# B&R Automation Studio project BatteryControl (part 4)

```iecst
	sustainHF[0]:=50.000;
	sustainHF[1]:=50.000;
	sustainHF[2]:=50.000;
	sustainHF[3]:=50.000;
	sustainHF[4]:=50.000;
	sustainHF[5]:=50.000;
	sustainHF[6]:=50.000;
	sustainHF[7]:=50.000;
	sustainHF[8]:=50.000;
	sustainHF[9]:=50.000;
	sustainHF[10]:=50.000;
	sustainHF[11]:=50.000;
	sustainHF[12]:=50.000;
	sustainHF[13]:=50.000;
	sustainHF[14]:=50.000;
	sustainHF[15]:=50.000;
	sustainHF[16]:=50.000;
	sustainHF[17]:=50.000;
	sustainHF[18]:=50.000;
	sustainHF[19]:=50.000;
	sustainHF[20]:=50.000;
	sustainHF[21]:=50.000;
	sustainHF[22]:=50.000;
	sustainHF[23]:=50.000;
	sustainHF[24]:=50.000;
	sustainHF[25]:=50.000;
	sustainHF[26]:=50.000;
	sustainHF[27]:=50.000;
	sustainHF[28]:=50.000;
	sustainHF[29]:=50.000;
	sustainHF[30]:=50.600;
	sustainHF[31]:=50.600;
	sustainHF[32]:=50.600;
	sustainHF[33]:=50.600;
	sustainHF[34]:=50.600;
	sustainHF[35]:=50.600;
	sustainHF[36]:=50.600;
	sustainHF[37]:=50.600;
	sustainHF[38]:=50.600;
	sustainHF[39]:=50.600;
	sustainHF[40]:=50.600;
	sustainHF[41]:=50.600;
	sustainHF[42]:=50.600;
	sustainHF[43]:=50.600;
	sustainHF[44]:=50.600;
	sustainHF[45]:=50.600;
	sustainHF[46]:=50.600;
	sustainHF[47]:=50.600;
	sustainHF[48]:=50.600;
	sustainHF[49]:=50.600;
	sustainHF[50]:=50.600;
	sustainHF[51]:=50.600;
	sustainHF[52]:=50.600;
	sustainHF[53]:=50.600;
	sustainHF[54]:=50.600;
	sustainHF[55]:=50.600;
	sustainHF[56]:=50.600;
	sustainHF[57]:=50.600;
	sustainHF[58]:=50.600;
	sustainHF[59]:=50.600;
	sustainHF[60]:=50.600;
	sustainHF[61]:=50.600;
	sustainHF[62]:=50.600;
	sustainHF[63]:=50.600;
	sustainHF[64]:=50.600;
	sustainHF[65]:=50.600;
	sustainHF[66]:=50.600;
	sustainHF[67]:=50.600;
	sustainHF[68]:=50.600;
	sustainHF[69]:=50.600;
	sustainHF[70]:=50.600;
	sustainHF[71]:=50.600;
	sustainHF[72]:=50.600;
	sustainHF[73]:=50.600;
	sustainHF[74]:=50.600;
	sustainHF[75]:=50.600;
	sustainHF[76]:=50.600;
	sustainHF[77]:=50.600;
	sustainHF[78]:=50.600;
	sustainHF[79]:=50.600;
	sustainHF[80]:=50.600;
	sustainHF[81]:=50.600;
	sustainHF[82]:=50.600;
	sustainHF[83]:=50.600;
	sustainHF[84]:=50.600;
	sustainHF[85]:=50.600;
	sustainHF[86]:=50.600;
	sustainHF[87]:=50.600;
	sustainHF[88]:=50.600;
	sustainHF[89]:=50.600;
	sustainHF[90]:=50.600;
	sustainHF[91]:=50.600;
	sustainHF[92]:=50.600;
	sustainHF[93]:=50.600;
	sustainHF[94]:=50.600;
	sustainHF[95]:=50.600;
	sustainHF[96]:=50.600;
	sustainHF[97]:=50.600;
	sustainHF[98]:=50.600;
	sustainHF[99]:=50.600;
	sustainHF[100]:=50.600;
	sustainHF[101]:=50.600;
	sustainHF[102]:=50.600;
	sustainHF[103]:=50.600;
	sustainHF[104]:=50.600;
	sustainHF[105]:=50.600;
	sustainHF[106]:=50.600;
	sustainHF[107]:=50.600;
	sustainHF[108]:=50.600;
	sustainHF[109]:=50.600;
	sustainHF[110]:=50.600;
	sustainHF[111]:=50.600;
	sustainHF[112]:=50.600;
	sustainHF[113]:=50.600;
	sustainHF[114]:=50.600;
	sustainHF[115]:=50.600;
	sustainHF[116]:=50.600;
	sustainHF[117]:=50.600;
	sustainHF[118]:=50.600;
	sustainHF[119]:=50.600;
	sustainHF[120]:=50.600;
	sustainHF[121]:=50.600;
	sustainHF[122]:=50.600;
	sustainHF[123]:=50.600;
	sustainHF[124]:=50.600;
	sustainHF[125]:=50.600;
	sustainHF[126]:=50.600;
	sustainHF[127]:=50.600;
	sustainHF[128]:=50.600;
	sustainHF[129]:=50.600;
	sustainHF[130]:=50.600;
	sustainHF[131]:=50.600;
	sustainHF[132]:=50.600;
	sustainHF[133]:=50.600;
	sustainHF[134]:=50.600;
	sustainHF[135]:=50.600;
	sustainHF[136]:=50.600;
	sustainHF[137]:=50.600;
	sustainHF[138]:=50.600;
	sustainHF[139]:=50.600;
	sustainHF[140]:=50.600;
	sustainHF[141]:=50.600;
	sustainHF[142]:=50.600;
	sustainHF[143]:=50.600;
	sustainHF[144]:=50.600;
	sustainHF[145]:=50.600;
	sustainHF[146]:=50.600;
	sustainHF[147]:=50.600;
	sustainHF[148]:=50.600;
	sustainHF[149]:=50.600;
	sustainHF[150]:=50.600;
	sustainHF[151]:=50.600;
	sustainHF[152]:=50.600;
	sustainHF[153]:=50.600;
	sustainHF[154]:=50.600;
	sustainHF[155]:=50.600;
	sustainHF[156]:=50.600;
	sustainHF[157]:=50.600;
	sustainHF[158]:=50.600;
	sustainHF[159]:=50.600;
	sustainHF[160]:=50.600;
	sustainHF[161]:=50.600;
	sustainHF[162]:=50.600;
	sustainHF[163]:=50.600;
	sustainHF[164]:=50.600;
	sustainHF[165]:=50.600;
	sustainHF[166]:=50.600;
	sustainHF[167]:=50.600;
	sustainHF[168]:=50.600;
	sustainHF[169]:=50.600;
	sustainHF[170]:=50.600;
	sustainHF[171]:=50.600;
	sustainHF[172]:=50.600;
	sustainHF[173]:=50.600;
	sustainHF[174]:=50.600;
	sustainHF[175]:=50.600;
	sustainHF[176]:=50.600;
	sustainHF[177]:=50.600;
	sustainHF[178]:=50.600;
	sustainHF[179]:=50.600;
	sustainHF[180]:=50.600;
	sustainHF[181]:=50.600;
	sustainHF[182]:=50.600;
	sustainHF[183]:=50.600;
	sustainHF[184]:=50.600;
	sustainHF[185]:=50.600;
	sustainHF[186]:=50.600;
	sustainHF[187]:=50.600;
	sustainHF[188]:=50.600;
	sustainHF[189]:=50.600;
	sustainHF[190]:=50.600;
	sustainHF[191]:=50.600;
	sustainHF[192]:=50.600;
	sustainHF[193]:=50.600;
	sustainHF[194]:=50.600;
	sustainHF[195]:=50.600;
	sustainHF[196]:=50.600;
	sustainHF[197]:=50.600;
	sustainHF[198]:=50.600;
	sustainHF[199]:=50.600;
	sustainHF[200]:=50.600;
	sustainHF[201]:=50.600;
	sustainHF[202]:=50.600;
	sustainHF[203]:=50.600;
	sustainHF[204]:=50.600;
	sustainHF[205]:=50.600;
	sustainHF[206]:=50.600;
	sustainHF[207]:=50.600;
	sustainHF[208]:=50.600;
	sustainHF[209]:=50.600;
	sustainHF[210]:=50.600;
	sustainHF[211]:=50.600;
	sustainHF[212]:=50.600;
	sustainHF[213]:=50.600;
	sustainHF[214]:=50.600;
	sustainHF[215]:=50.600;
	sustainHF[216]:=50.600;
	sustainHF[217]:=50.600;
	sustainHF[218]:=50.600;
	sustainHF[219]:=50.600;
	sustainHF[220]:=50.600;
	sustainHF[221]:=50.600;
	sustainHF[222]:=50.600;
	sustainHF[223]:=50.600;
	sustainHF[224]:=50.600;
	sustainHF[225]:=50.600;
	sustainHF[226]:=50.600;
	sustainHF[227]:=50.600;
	sustainHF[228]:=50.600;
	sustainHF[229]:=50.600;
	sustainHF[230]:=50.600;
	sustainHF[231]:=50.600;
	sustainHF[232]:=50.600;
	sustainHF[233]:=50.600;
	sustainHF[234]:=50.600;
	sustainHF[235]:=50.600;
	sustainHF[236]:=50.600;
	sustainHF[237]:=50.600;
	sustainHF[238]:=50.600;
	sustainHF[239]:=50.600;
	sustainHF[240]:=50.600;
	sustainHF[241]:=50.600;
	sustainHF[242]:=50.600;
	sustainHF[243]:=50.600;
	sustainHF[244]:=50.600;
	sustainHF[245]:=50.600;
	sustainHF[246]:=50.600;
	sustainHF[247]:=50.600;
	sustainHF[248]:=50.600;
	sustainHF[249]:=50.600;
	sustainHF[250]:=50.600;
	sustainHF[251]:=50.600;
	sustainHF[252]:=50.600;
	sustainHF[253]:=50.600;
	sustainHF[254]:=50.600;
	sustainHF[255]:=50.600;
	sustainHF[256]:=50.600;
	sustainHF[257]:=50.600;
	sustainHF[258]:=50.600;
	sustainHF[259]:=50.600;
	sustainHF[260]:=50.600;
	sustainHF[261]:=50.600;
	sustainHF[262]:=50.600;
	sustainHF[263]:=50.600;
	sustainHF[264]:=50.600;
	sustainHF[265]:=50.600;
	sustainHF[266]:=50.600;
	sustainHF[267]:=50.600;
	sustainHF[268]:=50.600;
	sustainHF[269]:=50.600;
	sustainHF[270]:=50.600;
	sustainHF[271]:=50.600;
	sustainHF[272]:=50.600;
	sustainHF[273]:=50.600;
	sustainHF[274]:=50.600;
	sustainHF[275]:=50.600;
	sustainHF[276]:=50.600;
	sustainHF[277]:=50.600;
	sustainHF[278]:=50.600;
	sustainHF[279]:=50.600;
	sustainHF[280]:=50.600;
	sustainHF[281]:=50.600;
	sustainHF[282]:=50.600;
	sustainHF[283]:=50.600;
	sustainHF[284]:=50.600;
	sustainHF[285]:=50.600;
	sustainHF[286]:=50.600;
	sustainHF[287]:=50.600;
	sustainHF[288]:=50.600;
	sustainHF[289]:=50.600;
	sustainHF[290]:=50.600;
	sustainHF[291]:=50.600;
	sustainHF[292]:=50.600;
	sustainHF[293]:=50.600;
	sustainHF[294]:=50.600;
	sustainHF[295]:=50.600;
	sustainHF[296]:=50.600;
	sustainHF[297]:=50.600;
	sustainHF[298]:=50.600;
	sustainHF[299]:=50.600;
	sustainHF[300]:=50.600;
	sustainHF[301]:=50.600;
	sustainHF[302]:=50.600;
	sustainHF[303]:=50.600;
	sustainHF[304]:=50.600;
	sustainHF[305]:=50.600;
	sustainHF[306]:=50.600;
	sustainHF[307]:=50.600;
	sustainHF[308]:=50.600;
	sustainHF[309]:=50.600;
	sustainHF[310]:=50.600;
	sustainHF[311]:=50.600;
	sustainHF[312]:=50.600;
	sustainHF[313]:=50.600;
	sustainHF[314]:=50.600;
	sustainHF[315]:=50.600;
	sustainHF[316]:=50.600;
	sustainHF[317]:=50.600;
	sustainHF[318]:=50.600;
	sustainHF[319]:=50.600;
	sustainHF[320]:=50.600;
	sustainHF[321]:=50.600;
	sustainHF[322]:=50.600;
	sustainHF[323]:=50.600;
	sustainHF[324]:=50.600;
	sustainHF[325]:=50.600;
	sustainHF[326]:=50.600;
	sustainHF[327]:=50.600;
	sustainHF[328]:=50.600;
	sustainHF[329]:=50.600;
	sustainHF[330]:=50.600;
	sustainHF[331]:=50.600;
	sustainHF[332]:=50.600;
	sustainHF[333]:=50.600;
	sustainHF[334]:=50.600;
	sustainHF[335]:=50.600;
	sustainHF[336]:=50.600;
	sustainHF[337]:=50.600;
	sustainHF[338]:=50.600;
	sustainHF[339]:=50.600;
	sustainHF[340]:=50.600;
	sustainHF[341]:=50.600;
	sustainHF[342]:=50.600;
	sustainHF[343]:=50.600;
	sustainHF[344]:=50.600;
	sustainHF[345]:=50.600;
	sustainHF[346]:=50.600;
	sustainHF[347]:=50.600;
	sustainHF[348]:=50.600;
	sustainHF[349]:=50.600;
	sustainHF[350]:=50.600;
	sustainHF[351]:=50.600;
	sustainHF[352]:=50.600;
	sustainHF[353]:=50.600;
	sustainHF[354]:=50.600;
	sustainHF[355]:=50.600;
	sustainHF[356]:=50.600;
	sustainHF[357]:=50.600;
	sustainHF[358]:=50.600;
	sustainHF[359]:=50.600;
	sustainHF[360]:=50.600;
	sustainHF[361]:=50.600;
	sustainHF[362]:=50.600;
	sustainHF[363]:=50.600;
	sustainHF[364]:=50.600;
	sustainHF[365]:=50.600;
	sustainHF[366]:=50.600;
	sustainHF[367]:=50.600;
	sustainHF[368]:=50.600;
	sustainHF[369]:=50.600;
	sustainHF[370]:=50.600;
	sustainHF[371]:=50.600;
	sustainHF[372]:=50.600;
	sustainHF[373]:=50.600;
	sustainHF[374]:=50.600;
	sustainHF[375]:=50.600;
	sustainHF[376]:=50.600;
	sustainHF[377]:=50.600;
	sustainHF[378]:=50.600;
	sustainHF[379]:=50.600;
	sustainHF[380]:=50.600;
	sustainHF[381]:=50.600;
	sustainHF[382]:=50.600;
	sustainHF[383]:=50.600;
	sustainHF[384]:=50.600;
	sustainHF[385]:=50.600;
	sustainHF[386]:=50.600;
	sustainHF[387]:=50.600;
	sustainHF[388]:=50.600;
	sustainHF[389]:=50.600;
	sustainHF[390]:=50.600;
	sustainHF[391]:=50.600;
	sustainHF[392]:=50.600;
	sustainHF[393]:=50.600;
	sustainHF[394]:=50.600;
	sustainHF[395]:=50.600;
	sustainHF[396]:=50.600;
	sustainHF[397]:=50.600;
	sustainHF[398]:=50.600;
	sustainHF[399]:=50.600;
	sustainHF[400]:=50.600;
	sustainHF[401]:=50.600;
	sustainHF[402]:=50.600;
	sustainHF[403]:=50.600;
	sustainHF[404]:=50.600;
	sustainHF[405]:=50.600;
	sustainHF[406]:=50.600;
	sustainHF[407]:=50.600;
	sustainHF[408]:=50.600;
	sustainHF[409]:=50.600;
	sustainHF[410]:=50.600;
	sustainHF[411]:=50.600;
	sustainHF[412]:=50.600;
	sustainHF[413]:=50.600;
	sustainHF[414]:=50.600;
	sustainHF[415]:=50.600;
	sustainHF[416]:=50.600;
	sustainHF[417]:=50.600;
	sustainHF[418]:=50.600;
	sustainHF[419]:=50.600;
	sustainHF[420]:=50.600;
	sustainHF[421]:=50.600;
	sustainHF[422]:=50.600;
	sustainHF[423]:=50.600;
	sustainHF[424]:=50.600;
	sustainHF[425]:=50.600;
	sustainHF[426]:=50.600;
	sustainHF[427]:=50.600;
	sustainHF[428]:=50.600;
	sustainHF[429]:=50.600;
	sustainHF[430]:=50.600;
	sustainHF[431]:=50.600;
	sustainHF[432]:=50.600;
	sustainHF[433]:=50.600;
	sustainHF[434]:=50.600;
	sustainHF[435]:=50.600;
	sustainHF[436]:=50.600;
	sustainHF[437]:=50.600;
	sustainHF[438]:=50.600;
	sustainHF[439]:=50.600;
	sustainHF[440]:=50.600;
	sustainHF[441]:=50.600;
	sustainHF[442]:=50.600;
	sustainHF[443]:=50.600;
	sustainHF[444]:=50.600;
	sustainHF[445]:=50.600;
	sustainHF[446]:=50.600;
	sustainHF[447]:=50.600;
	sustainHF[448]:=50.600;
	sustainHF[449]:=50.600;
	sustainHF[450]:=50.600;
	sustainHF[451]:=50.600;
	sustainHF[452]:=50.600;
	sustainHF[453]:=50.600;
	sustainHF[454]:=50.600;
	sustainHF[455]:=50.600;
	sustainHF[456]:=50.600;
	sustainHF[457]:=50.600;
	sustainHF[458]:=50.600;
	sustainHF[459]:=50.600;
	sustainHF[460]:=50.600;
	sustainHF[461]:=50.600;
	sustainHF[462]:=50.600;
	sustainHF[463]:=50.600;
	sustainHF[464]:=50.600;
	sustainHF[465]:=50.600;
	sustainHF[466]:=50.600;
	sustainHF[467]:=50.600;
	sustainHF[468]:=50.600;
	sustainHF[469]:=50.600;
	sustainHF[470]:=50.600;
	sustainHF[471]:=50.600;
	sustainHF[472]:=50.600;
	sustainHF[473]:=50.600;
	sustainHF[474]:=50.600;
	sustainHF[475]:=50.600;
	sustainHF[476]:=50.600;
	sustainHF[477]:=50.600;
	sustainHF[478]:=50.600;
	sustainHF[479]:=50.600;
	sustainHF[480]:=50.600;
	sustainHF[481]:=50.600;
	sustainHF[482]:=50.600;
	sustainHF[483]:=50.600;
	sustainHF[484]:=50.600;
	sustainHF[485]:=50.600;
	sustainHF[486]:=50.600;
	sustainHF[487]:=50.600;
	sustainHF[488]:=50.600;
	sustainHF[489]:=50.600;
	sustainHF[490]:=50.600;
	sustainHF[491]:=50.600;
	sustainHF[492]:=50.600;
	sustainHF[493]:=50.600;
	sustainHF[494]:=50.600;
	sustainHF[495]:=50.600;
	sustainHF[496]:=50.600;
	sustainHF[497]:=50.600;
	sustainHF[498]:=50.600;
	sustainHF[499]:=50.600;
	sustainHF[500]:=50.600;
	sustainHF[501]:=50.600;
	sustainHF[502]:=50.600;
	sustainHF[503]:=50.600;
	sustainHF[504]:=50.600;
	sustainHF[505]:=50.600;
	sustainHF[506]:=50.600;
	sustainHF[507]:=50.600;
	sustainHF[508]:=50.600;
	sustainHF[509]:=50.600;
	sustainHF[510]:=50.600;
	sustainHF[511]:=50.600;
	sustainHF[512]:=50.600;
	sustainHF[513]:=50.600;
	sustainHF[514]:=50.600;
	sustainHF[515]:=50.600;
	sustainHF[516]:=50.600;
	sustainHF[517]:=50.600;
	sustainHF[518]:=50.600;
	sustainHF[519]:=50.600;
	sustainHF[520]:=50.600;
	sustainHF[521]:=50.600;
	sustainHF[522]:=50.600;
	sustainHF[523]:=50.600;
	sustainHF[524]:=50.600;
	sustainHF[525]:=50.600;
	sustainHF[526]:=50.600;
	sustainHF[527]:=50.600;
	sustainHF[528]:=50.600;
	sustainHF[529]:=50.600;
	sustainHF[530]:=50.600;
	sustainHF[531]:=50.600;
	sustainHF[532]:=50.600;
	sustainHF[533]:=50.600;
	sustainHF[534]:=50.600;
	sustainHF[535]:=50.600;
	sustainHF[536]:=50.600;
	sustainHF[537]:=50.600;
	sustainHF[538]:=50.600;
	sustainHF[539]:=50.600;
	sustainHF[540]:=50.600;
	sustainHF[541]:=50.600;
	sustainHF[542]:=50.600;
	sustainHF[543]:=50.600;
	sustainHF[544]:=50.600;
	sustainHF[545]:=50.600;
	sustainHF[546]:=50.600;
	sustainHF[547]:=50.600;
	sustainHF[548]:=50.600;
	sustainHF[549]:=50.600;
	sustainHF[550]:=50.600;
	sustainHF[551]:=50.600;
	sustainHF[552]:=50.600;
	sustainHF[553]:=50.600;
	sustainHF[554]:=50.600;
	sustainHF[555]:=50.600;
	sustainHF[556]:=50.600;
	sustainHF[557]:=50.600;
	sustainHF[558]:=50.600;
	sustainHF[559]:=50.600;
	sustainHF[560]:=50.600;
	sustainHF[561]:=50.600;
	sustainHF[562]:=50.600;
	sustainHF[563]:=50.600;
	sustainHF[564]:=50.600;
	sustainHF[565]:=50.600;
	sustainHF[566]:=50.600;
	sustainHF[567]:=50.600;
	sustainHF[568]:=50.600;
	sustainHF[569]:=50.600;
	sustainHF[570]:=50.600;
	sustainHF[571]:=50.600;
	sustainHF[572]:=50.600;
	sustainHF[573]:=50.600;
	sustainHF[574]:=50.600;
	sustainHF[575]:=50.600;
	sustainHF[576]:=50.600;
	sustainHF[577]:=50.600;
	sustainHF[578]:=50.600;
	sustainHF[579]:=50.600;
	sustainHF[580]:=50.600;
	sustainHF[581]:=50.600;
	sustainHF[582]:=50.600;
	sustainHF[583]:=50.600;
	sustainHF[584]:=50.600;
	sustainHF[585]:=50.600;
	sustainHF[586]:=50.600;
	sustainHF[587]:=50.600;
	sustainHF[588]:=50.600;
	sustainHF[589]:=50.600;
	sustainHF[590]:=50.600;
	sustainHF[591]:=50.600;
	sustainHF[592]:=50.600;
	sustainHF[593]:=50.600;
	sustainHF[594]:=50.600;
	sustainHF[595]:=50.600;
	sustainHF[596]:=50.600;
	sustainHF[597]:=50.600;
	sustainHF[598]:=50.600;
	sustainHF[599]:=50.600;
	sustainHF[600]:=50.600;
	sustainHF[601]:=50.600;
	sustainHF[602]:=50.600;
	sustainHF[603]:=50.600;
	sustainHF[604]:=50.600;
	sustainHF[605]:=50.600;
	sustainHF[606]:=50.600;
	sustainHF[607]:=50.600;
	sustainHF[608]:=50.600;
	sustainHF[609]:=50.600;
	sustainHF[610]:=50.600;
	sustainHF[611]:=50.600;
	sustainHF[612]:=50.600;
	sustainHF[613]:=50.600;
	sustainHF[614]:=50.600;
	sustainHF[615]:=50.600;
	sustainHF[616]:=50.600;
	sustainHF[617]:=50.600;
	sustainHF[618]:=50.600;
	sustainHF[619]:=50.600;
	sustainHF[620]:=50.600;
	sustainHF[621]:=50.600;
	sustainHF[622]:=50.600;
	sustainHF[623]:=50.600;
	sustainHF[624]:=50.600;
	sustainHF[625]:=50.600;
	sustainHF[626]:=50.600;
	sustainHF[627]:=50.600;
	sustainHF[628]:=50.600;
	sustainHF[629]:=50.600;
	sustainHF[630]:=50.600;
	sustainHF[631]:=50.600;
	sustainHF[632]:=50.600;
	sustainHF[633]:=50.600;
	sustainHF[634]:=50.600;
	sustainHF[635]:=50.600;
	sustainHF[636]:=50.600;
	sustainHF[637]:=50.600;
	sustainHF[638]:=50.600;
	sustainHF[639]:=50.600;
	sustainHF[640]:=50.600;
	sustainHF[641]:=50.600;
	sustainHF[642]:=50.600;
	sustainHF[643]:=50.600;
	sustainHF[644]:=50.600;
	sustainHF[645]:=50.600;
	sustainHF[646]:=50.600;
	sustainHF[647]:=50.600;
	sustainHF[648]:=50.600;
	sustainHF[649]:=50.600;
	sustainHF[650]:=50.600;
	sustainHF[651]:=50.600;
	sustainHF[652]:=50.600;
	sustainHF[653]:=50.600;
	sustainHF[654]:=50.600;
	sustainHF[655]:=50.600;
	sustainHF[656]:=50.600;
	sustainHF[657]:=50.600;
	sustainHF[658]:=50.600;
	sustainHF[659]:=50.600;
	sustainHF[660]:=50.600;
	sustainHF[661]:=50.600;
	sustainHF[662]:=50.600;
	sustainHF[663]:=50.600;
	sustainHF[664]:=50.600;
	sustainHF[665]:=50.600;
	sustainHF[666]:=50.600;
	sustainHF[667]:=50.600;
	sustainHF[668]:=50.600;
	sustainHF[669]:=50.600;
	sustainHF[670]:=50.600;
	sustainHF[671]:=50.600;
	sustainHF[672]:=50.600;
	sustainHF[673]:=50.600;
	sustainHF[674]:=50.600;
	sustainHF[675]:=50.600;
	sustainHF[676]:=50.600;
	sustainHF[677]:=50.600;
	sustainHF[678]:=50.600;
	sustainHF[679]:=50.600;
	sustainHF[680]:=50.600;
	sustainHF[681]:=50.600;
	sustainHF[682]:=50.600;
	sustainHF[683]:=50.600;
	sustainHF[684]:=50.600;
	sustainHF[685]:=50.600;
	sustainHF[686]:=50.600;
	sustainHF[687]:=50.600;
	sustainHF[688]:=50.600;
	sustainHF[689]:=50.600;
	sustainHF[690]:=50.600;
	sustainHF[691]:=50.600;
	sustainHF[692]:=50.600;
	sustainHF[693]:=50.600;
	sustainHF[694]:=50.600;
	sustainHF[695]:=50.600;
	sustainHF[696]:=50.600;
	sustainHF[697]:=50.600;
	sustainHF[698]:=50.600;
	sustainHF[699]:=50.600;
	sustainHF[700]:=50.600;
	sustainHF[701]:=50.600;
	sustainHF[702]:=50.600;
	sustainHF[703]:=50.600;
	sustainHF[704]:=50.600;
	sustainHF[705]:=50.600;
	sustainHF[706]:=50.600;
	sustainHF[707]:=50.600;
	sustainHF[708]:=50.600;
	sustainHF[709]:=50.600;
	sustainHF[710]:=50.600;
	sustainHF[711]:=50.600;
	sustainHF[712]:=50.600;
	sustainHF[713]:=50.600;
	sustainHF[714]:=50.600;
	sustainHF[715]:=50.600;
	sustainHF[716]:=50.600;
	sustainHF[717]:=50.600;
	sustainHF[718]:=50.600;
	sustainHF[719]:=50.600;
	sustainHF[720]:=50.600;
	sustainHF[721]:=50.600;
	sustainHF[722]:=50.600;
	sustainHF[723]:=50.600;
	sustainHF[724]:=50.600;
	sustainHF[725]:=50.600;
	sustainHF[726]:=50.600;
	sustainHF[727]:=50.600;
	sustainHF[728]:=50.600;
	sustainHF[729]:=50.600;
	sustainHF[730]:=50.600;
	sustainHF[731]:=50.600;
	sustainHF[732]:=50.600;
	sustainHF[733]:=50.600;
	sustainHF[734]:=50.600;
	sustainHF[735]:=50.600;
	sustainHF[736]:=50.600;
	sustainHF[737]:=50.600;
	sustainHF[738]:=50.600;
	sustainHF[739]:=50.600;
	sustainHF[740]:=50.600;
	sustainHF[741]:=50.600;
	sustainHF[742]:=50.600;
	sustainHF[743]:=50.600;
	sustainHF[744]:=50.600;
	sustainHF[745]:=50.600;
	sustainHF[746]:=50.600;
	sustainHF[747]:=50.600;
	sustainHF[748]:=50.600;
	sustainHF[749]:=50.600;
	sustainHF[750]:=50.600;
	sustainHF[751]:=50.600;
	sustainHF[752]:=50.600;
	sustainHF[753]:=50.600;
	sustainHF[754]:=50.600;
	sustainHF[755]:=50.600;
	sustainHF[756]:=50.600;
	sustainHF[757]:=50.600;
	sustainHF[758]:=50.600;
	sustainHF[759]:=50.600;
	sustainHF[760]:=50.600;
	sustainHF[761]:=50.600;
	sustainHF[762]:=50.600;
	sustainHF[763]:=50.600;
	sustainHF[764]:=50.600;
	sustainHF[765]:=50.600;
	sustainHF[766]:=50.600;
	sustainHF[767]:=50.600;
	sustainHF[768]:=50.600;
	sustainHF[769]:=50.600;
	sustainHF[770]:=50.600;
	sustainHF[771]:=50.600;
	sustainHF[772]:=50.600;
	sustainHF[773]:=50.600;
	sustainHF[774]:=50.600;
	sustainHF[775]:=50.600;
	sustainHF[776]:=50.600;
	sustainHF[777]:=50.600;
	sustainHF[778]:=50.600;
	sustainHF[779]:=50.600;
	sustainHF[780]:=50.600;
	sustainHF[781]:=50.600;
	sustainHF[782]:=50.600;
	sustainHF[783]:=50.600;
	sustainHF[784]:=50.600;
	sustainHF[785]:=50.600;
	sustainHF[786]:=50.600;
	sustainHF[787]:=50.600;
	sustainHF[788]:=50.600;
	sustainHF[789]:=50.600;
	sustainHF[790]:=50.600;
	sustainHF[791]:=50.600;
	sustainHF[792]:=50.600;
	sustainHF[793]:=50.600;
	sustainHF[794]:=50.600;
	sustainHF[795]:=50.600;
	sustainHF[796]:=50.600;
	sustainHF[797]:=50.600;
	sustainHF[798]:=50.600;
	sustainHF[799]:=50.600;
	sustainHF[800]:=50.600;
	sustainHF[801]:=50.600;
	sustainHF[802]:=50.600;
	sustainHF[803]:=50.600;
	sustainHF[804]:=50.600;
	sustainHF[805]:=50.600;
	sustainHF[806]:=50.600;
	sustainHF[807]:=50.600;
	sustainHF[808]:=50.600;
	sustainHF[809]:=50.600;
	sustainHF[810]:=50.600;
	sustainHF[811]:=50.600;
	sustainHF[812]:=50.600;
	sustainHF[813]:=50.600;
	sustainHF[814]:=50.600;
	sustainHF[815]:=50.600;
	sustainHF[816]:=50.600;
	sustainHF[817]:=50.600;
	sustainHF[818]:=50.600;
	sustainHF[819]:=50.600;
	sustainHF[820]:=50.600;
	sustainHF[821]:=50.600;
	sustainHF[822]:=50.600;
	sustainHF[823]:=50.600;
	sustainHF[824]:=50.600;
	sustainHF[825]:=50.600;
	sustainHF[826]:=50.600;
	sustainHF[827]:=50.600;
	sustainHF[828]:=50.600;
	sustainHF[829]:=50.600;
	sustainHF[830]:=50.600;
	sustainHF[831]:=50.600;
	sustainHF[832]:=50.600;
	sustainHF[833]:=50.600;
	sustainHF[834]:=50.600;
	sustainHF[835]:=50.600;
	sustainHF[836]:=50.600;
	sustainHF[837]:=50.600;
	sustainHF[838]:=50.600;
	sustainHF[839]:=50.600;
	sustainHF[840]:=50.600;
	sustainHF[841]:=50.600;
	sustainHF[842]:=50.600;
	sustainHF[843]:=50.600;
	sustainHF[844]:=50.600;
	sustainHF[845]:=50.600;
	sustainHF[846]:=50.600;
	sustainHF[847]:=50.600;
	sustainHF[848]:=50.600;
	sustainHF[849]:=50.600;
	sustainHF[850]:=50.600;
	sustainHF[851]:=50.600;
	sustainHF[852]:=50.600;
	sustainHF[853]:=50.600;
	sustainHF[854]:=50.600;
	sustainHF[855]:=50.600;
	sustainHF[856]:=50.600;
	sustainHF[857]:=50.600;
	sustainHF[858]:=50.600;
	sustainHF[859]:=50.600;
	sustainHF[860]:=50.600;
	sustainHF[861]:=50.600;
	sustainHF[862]:=50.600;
	sustainHF[863]:=50.600;
	sustainHF[864]:=50.600;
	sustainHF[865]:=50.600;
	sustainHF[866]:=50.600;
	sustainHF[867]:=50.600;
	sustainHF[868]:=50.600;
	sustainHF[869]:=50.600;
	sustainHF[870]:=50.600;
	sustainHF[871]:=50.600;
	sustainHF[872]:=50.600;
	sustainHF[873]:=50.600;
	sustainHF[874]:=50.600;
	sustainHF[875]:=50.600;
	sustainHF[876]:=50.600;
	sustainHF[877]:=50.600;
	sustainHF[878]:=50.600;
	sustainHF[879]:=50.600;
	sustainHF[880]:=50.600;
	sustainHF[881]:=50.600;
	sustainHF[882]:=50.600;
	sustainHF[883]:=50.600;
	sustainHF[884]:=50.600;
	sustainHF[885]:=50.600;
	sustainHF[886]:=50.600;
	sustainHF[887]:=50.600;
	sustainHF[888]:=50.600;
	sustainHF[889]:=50.600;
	sustainHF[890]:=50.600;
	sustainHF[891]:=50.600;
	sustainHF[892]:=50.600;
	sustainHF[893]:=50.600;
	sustainHF[894]:=50.600;
	sustainHF[895]:=50.600;
	sustainHF[896]:=50.600;
	sustainHF[897]:=50.600;
	sustainHF[898]:=50.600;
	sustainHF[899]:=50.600;
	sustainHF[900]:=50.600;
	sustainHF[901]:=50.600;
	sustainHF[902]:=50.600;
	sustainHF[903]:=50.600;
	sustainHF[904]:=50.600;
	sustainHF[905]:=50.600;
	sustainHF[906]:=50.600;
	sustainHF[907]:=50.600;
	sustainHF[908]:=50.600;
	sustainHF[909]:=50.600;
	sustainHF[910]:=50.600;
	sustainHF[911]:=50.600;
	sustainHF[912]:=50.600;
	sustainHF[913]:=50.600;
	sustainHF[914]:=50.600;
	sustainHF[915]:=50.600;
	sustainHF[916]:=50.600;
	sustainHF[917]:=50.600;
	sustainHF[918]:=50.600;
	sustainHF[919]:=50.600;
	sustainHF[920]:=50.600;
	sustainHF[921]:=50.600;
	sustainHF[922]:=50.600;
	sustainHF[923]:=50.600;
	sustainHF[924]:=50.600;
	sustainHF[925]:=50.600;
	sustainHF[926]:=50.600;
	sustainHF[927]:=50.600;
	sustainHF[928]:=50.600;
	sustainHF[929]:=50.600;
	sustainHF[930]:=50.000;
	sustainHF[931]:=50.000;
	sustainHF[932]:=50.000;
	sustainHF[933]:=50.000;
	sustainHF[934]:=50.000;
	sustainHF[935]:=50.000;
	sustainHF[936]:=50.000;
	sustainHF[937]:=50.000;
	sustainHF[938]:=50.000;
	sustainHF[939]:=50.000;
	sustainHF[940]:=50.000;
	sustainHF[941]:=50.000;
	sustainHF[942]:=50.000;
	sustainHF[943]:=50.000;
	sustainHF[944]:=50.000;
	sustainHF[945]:=50.000;
	sustainHF[946]:=50.000;
	sustainHF[947]:=50.000;
	sustainHF[948]:=50.000;
	sustainHF[949]:=50.000;
	sustainHF[950]:=50.000;
	sustainHF[951]:=50.000;
	sustainHF[952]:=50.000;
	sustainHF[953]:=50.000;
	sustainHF[954]:=50.000;
	sustainHF[955]:=50.000;
	sustainHF[956]:=50.000;
	sustainHF[957]:=50.000;
	sustainHF[958]:=50.000;
	sustainHF[959]:=50.000;

END_PROGRAM
```

### Program Logical/Baseline (IEC)

#### Variables.var
```iecst
VAR
	status_gettime : UINT;
	rtc_gettime : RTCtime_typ;
	currentSP : INT;
	prevSP : INT;
	baselineSP : ARRAY[0..3] OF INT;
	Extra_Charge_SP : INT;
	Const_Charge_SP : INT;
	BaselineRamp : LCRampLim;
	NG_Charge_SP : INT;
	NG_SoC : UINT;
	Extra_Charge_SoC : UINT;
	Base_Charge_SoC : UINT;
	Local_DCadjMan : INT;
END_VAR
```

#### Cyclic.st
```iecst
PROGRAM _CYCLIC
	//get current time
	status_gettime := RTC_gettime(ADR(rtc_gettime));

	// get current SP
	IF rtc_gettime.minute >= 0 AND rtc_gettime.minute < 30 THEN
		currentSP := 1+2*rtc_gettime.hour;
	ELSE
		currentSP := 1+2*rtc_gettime.hour+1;
	END_IF;

	NG_Charge_SP := REAL_TO_INT(INT_TO_REAL(maxExpectedOutput) * 0.05 * -1);

	//when new SP
	IF currentSP <> prevSP THEN
		//shift baselines
	//	baselineSP[0] := baselineSP[1];
	//	baselineSP[1] := baselineSP[2];
	//	baselineSP[2] := baselineSP[3];

		//select the new baseline based on SoC
		IF RTACSoC < NG_SoC THEN
			baselineSP[0] := NG_Charge_SP;
		ELSIF RTACSoC < Extra_Charge_SoC THEN
			baselineSP[0] := Extra_Charge_SP;
		ELSIF  RTACSoC < Base_Charge_SoC THEN
			baselineSP[0] := Const_Charge_SP;
		ELSE
			baselineSP[0] := 0;
		END_IF;

		prevSP := currentSP;
	END_IF;

	//ramping of the baseline
	IF baselineAuto THEN
		BaselineRamp.x        := 	baselineSP[0]; //current baseline setting
	ELSE
		BaselineRamp.x := DCbaselineAdjustmentManual;
		DCbaselineAdjustmentManual := Local_DCadjMan;
	END_IF;

	BaselineRamp.basetime := baseLCCounter.seccnt;
	BaselineRamp();		(* LCRampLim function block call *)
	DCbaselineAdjustment := BaselineRamp.y; //output to DC algorythm

END_PROGRAM
```

#### Init.st
```iecst
PROGRAM _INIT
	BaselineRamp.enable    := TRUE;
	BaselineRamp.tup       := 2400;
	BaselineRamp.tdown     := 2400;
	BaselineRamp.max_value := maxExpectedOutput;
	BaselineRamp.min_value := -1*maxExpectedOutput;
	BaselineRamp.yset      := 0;
	BaselineRamp.set       := FALSE;

	baselineSP[0] := 0;
	baselineSP[1] := 0;
	baselineSP[2] := 0;
	baselineSP[3] := 0;

	baselineAuto := TRUE;

	prevSP := 0;

	NG_SoC := 280; //1/10
	Extra_Charge_SoC := 350; //1/10;
	Base_Charge_SoC := 450; //1/10;

	NG_Charge_SP := REAL_TO_INT(INT_TO_REAL(maxExpectedOutput) * 0.05);
	Extra_Charge_SP := -500;
	Const_Charge_SP := -100;

END_PROGRAM
```

### Program Logical/DNO_SIGNALS (IEC)

#### Cyclic.ab - Cyclic code
```automation-basic
PROGRAM _CYCLIC
	(* Insert code here *)
	IF Stage1_Input THEN				(* K1 is Stage 1 Confirm *)
		Stage1_Output := TRUE;			(* K3 is Stage 1 Enable *)
	ENDIF								(* K2 Is stage 2 Confirm *)
										(* K4 is Stage 2 Enable*)
										(* K5 is G59 Event *)
	IF Stage1_Input = FALSE THEN 		(* K6 is TX1&2 2&3 5&6 Feeder OPEN *)
		Stage1_Output := FALSE;
	ENDIF

	IF Stage1_Output THEN
		Stage1_Confirmed := TRUE;

	ENDIF

	IF Stage1_Output = FALSE THEN
		Stage1_Confirmed := FALSE;
		ENDIF

	IF Stage2_Input = TRUE AND TX123OPEN = TRUE THEN
		Stage2_Output:= TRUE;
	ENDIF

	IF Stage2_Output THEN
		Stage2_Confirmed:= TRUE;

	ENDIF
	IF TX123OPEN = FALSE THEN
		Stage2_Output := FALSE;
	ENDIF

	IF Stage2_Input = FALSE THEN
		Stage2_Output := FALSE;
	ENDIF

	IF Stage2_Output = FALSE THEN
		Stage2_Confirmed := FALSE;
	ENDIF

	TON_10ms(Stage2_Input AND NOT TX123OPEN, 1000, BreakerNotOpenAlarm, ElapsedTime);

END_PROGRAM
```

#### Init.ab - Init code
```automation-basic
PROGRAM _INIT
	(* Insert code here *)
	Stage1_Input := 0;
	Stage2_Input := 0;

END_PROGRAM
```

#### Variables.var - Local variables
```iecst
VAR
	Stage1_Input : BOOL;
	Stage2_Input : BOOL;
	G59_Input : BOOL;
	Stage1_Confirmed : BOOL;
	Stage2_Confirmed : BOOL;
	Stage1_Output : BOOL;
	Stage2_Output : BOOL;
	TX123OPEN : BOOL; (*TXFeeder123Open*)
	BreakerNotOpenAlarm : BOOL;
	ElapsedTime : UDINT;
END_VAR
```

### Program Logical/Watchdog (IEC)

#### Variables.var
```iecst
VAR
	Watchdog_Int : INT;
END_VAR
```

#### Cyclic.ab
```automation-basic
PROGRAM _CYCLIC
	(* Insert code here *)
Watchdog_Int := Watchdog_Int +1;

	IF Watchdog_Int = 10 THEN
		Watchdog_Int :=0;
		ENDIF
END_PROGRAM
```

#### Init.ab
```automation-basic
PROGRAM _INIT
	(* Insert code here *)

	Watchdog_Int = 0;

END_PROGRAM
```

- Visualisation Logical/mappView (not shown)

### Program Logical/DynamicContAll_BatLane

#### Variables.var
```iecst
VAR
	Table : MTLookUpTable;
	mtCONSTANT_END_VALUE : MTLookUpModeEnum;
	freqDev : REAL;
	powerOut : REAL;
	powerRatio : REAL;
	MAX_INJ_FREQ : UINT;
	MIN_INJ_FREQ : UINT;
END_VAR
VAR CONSTANT
	GRID_DEADAND : REAL := 0.015;
END_VAR
VAR
	freqDevUINT : UINT;
	freqDevINT : INT;
	prevPowerOutput : DINT;
	MovingAverage : MTFilterMovingAverage;
	expected : INT;
	diff : INT;
	powerOutputTmp : INT;
	error : REAL;
	LowPassFilter : MTFilterLowPass;
	mtBESSEL : MTFilterTypeEnum;
	filterFreqMA : REAL;
	filterFreqLowPass : REAL;
END_VAR
```

#### Cyclic.st
```iecst
PROGRAM _CYCLIC

	IF testModeOn THEN

		IF injFrequency < MIN_INJ_FREQ THEN
			injFrequency := MIN_INJ_FREQ;
		END_IF;

		IF injFrequency > MAX_INJ_FREQ THEN
			injFrequency := MAX_INJ_FREQ;
		END_IF;

	//	:= injFrequency;
	ELSE
		frequency := aiFrequency;
	END_IF;

	MovingAverage.In:= UINT_TO_REAL(frequency);
	MovingAverage();

	filterFreq := brmceil(MovingAverage.Out*10)/1000;
	filterFreqMA := brmceil(MovingAverage.Out*10)/1000;

	LowPassFilter.In:= UINT_TO_REAL(frequency);;
	LowPassFilter();

	filterFreqLowPass:= brmceil(LowPassFilter.Out*10)/1000;

	IF DynamicContainmentEnabled THEN

		IF NOT(diPhase1LossGen) THEN
			freqDev := filterFreq - GRID_FREQUENCY;
		ELSE
			freqDev := 0;
		END_IF;

		Table.InX:= freqDev;   (* freq deviation *)
		Table();          (* run table lookup *)
		powerRatio:= Table.Out; (* calculated % output *)

		powerOutputTmp :=  REAL_TO_INT(INT_TO_REAL(maxExpectedOutput) * powerRatio/100.00 + DCbaselineAdjustment);

		diff := expected - powerOutputTmp;

		error := (INT_TO_REAL(powerOutputTmp) / INT_TO_REAL(expected))*100 - 100;

		powerOutputDINT := REAL_TO_DINT(INT_TO_REAL(maxExpectedOutput) * powerRatio/100.00 + DCbaselineAdjustment);

		IF powerOutputDINT = 20000 THEN
			powerOutputDINT := 20200;
		END_IF;

	END_IF;

	IF NOT(cmdWritePowerOutput) AND NOT(WritePowerOutputACK) THEN

		IF prevPowerOutput <> powerOutputDINT THEN
			cmdWritePowerOutput := TRUE;
		END_IF;
		prevPowerOutput := powerOutputDINT;
	END_IF;

	IF WritePowerOutputACK THEN
		cmdWritePowerOutput := FALSE;
	END_IF;

END_PROGRAM
```

#### Init.st
```iecst
PROGRAM _INIT

    (* 1D lookup table *)
	Table.NodeVectorX[0] := -0.5;					Table.FcnValues[0] := 100;
	Table.NodeVectorX[1] := -0.2;					Table.FcnValues[1] := 5;
	Table.NodeVectorX[2] := -1*0.02;		Table.FcnValues[2] := 0.135;
	Table.NodeVectorX[3] := -1*GRID_DEADAND+0.001;	Table.FcnValues[3] := 0;
	Table.NodeVectorX[4] := GRID_DEADAND-0.001;		Table.FcnValues[4] := 0;
	//LF & HF
//	Table.NodeVectorX[5] := 0.02;					Table.FcnValues[5] := -0.135;
//	Table.NodeVectorX[6] := 0.2;					Table.FcnValues[6] := -5;
//	Table.NodeVectorX[7] := 0.5;					Table.FcnValues[7] := -100;

	//LF Only
	Table.NodeVectorX[5] := 0.02;			Table.FcnValues[5] := 0;
	Table.NodeVectorX[6] := 0.2;					Table.FcnValues[6] := 0;
	Table.NodeVectorX[7] := 0.5;					Table.FcnValues[7] := 0;

	Table.NumberOfNodes:= 8;
	Table.Mode:= mtCONSTANT_END_VALUE;
	Table.Enable:= 1; (* enable function block *)

	MAX_INJ_FREQ := 5200;
	MIN_INJ_FREQ := 4800;

	MovingAverage.WindowLength:= 3; (* moving window length *)
	MovingAverage.Enable:= 1;

	LowPassFilter.CutOffFrequency:= 20; (* cut-off frequency [Hz] *)
	LowPassFilter.Order:= 1;             (* 3rd order low-pass filter *)
	LowPassFilter.Type:= mtBESSEL;       (* bessel filter *)
	LowPassFilter.Enable:= 1;            (* enable function block *)

	DCbaselineAdjustment := 0;

	expected := 0;

	activePower := 0;

END_PROGRAM
```

Listed in the project but not available here: Logical/Global.typ, Logical/Modbus/Exit.st, Logical/Modbus/Types.typ, Logical/DNO_SIGNALS/Exit.ab, Logical/DNO_SIGNALS/Types.typ
